// Mitsubishi GX Works2 project: punya asisten   PLC: Q03UDV

PROGRAM MAIN
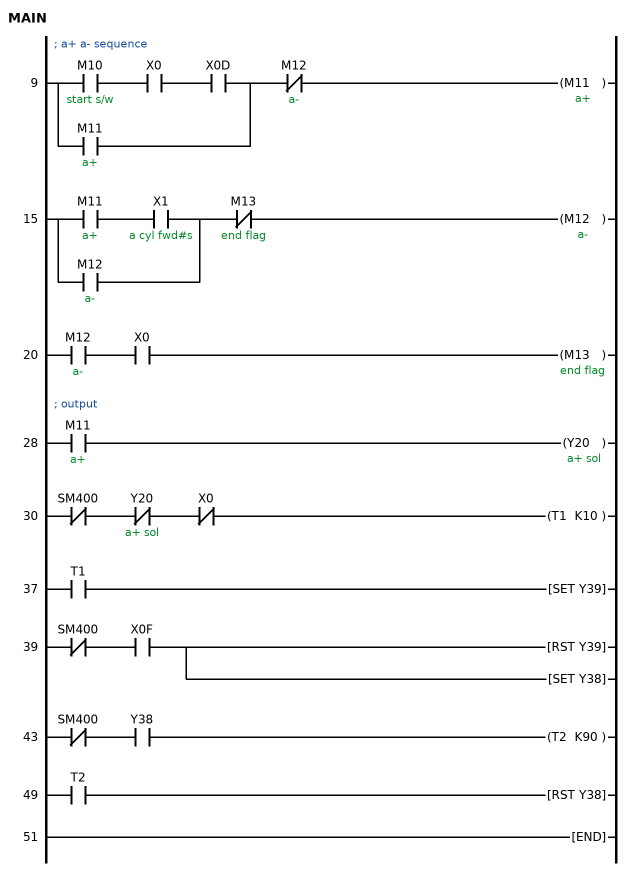
; a+ a- sequence
9     LD      M10  ; start s/w
      AND     X0
      AND     X0D
      OR      M11  ; a+
      ANI     M12  ; a-
      OUT     M11  ; a+
15    LD      M11  ; a+
      AND     X1  ; a cyl fwd#s
      OR      M12  ; a-
      ANI     M13  ; end flag
      OUT     M12  ; a-
20    LD      M12  ; a-
      AND     X0
      OUT     M13  ; end flag
; output
28    LD      M11  ; a+
      OUT     Y20  ; a+ sol
30    LDI     SM400
      ANI     Y20  ; a+ sol
      ANI     X0
      OUT     T1 K10
37    LD      T1
      SET     Y39
39    LDI     SM400
      AND     X0F
      RST     Y39
      SET     Y38
43    LDI     SM400
      AND     Y38
      OUT     T2 K90
49    LD      T2
      RST     Y38
51    END
END_PROGRAM

// device comments not shown above
M1000  ; end flag
